// TIA Portal V21 export
VAR_GLOBAL   // PLC tag table "ControlloVuotoReciveDigitali"
END_VAR
VAR_GLOBAL CONSTANT   // user constants
   K_SegnaleDaControlloVuoto_Allarme : Int := 1;
END_VAR
